FUNCTION fSHDLCChecksum : BYTE
VAR_INPUT
	i_bAdr	:	BYTE;
	i_bCmd	:	BYTE;
	i_bLen	:	BYTE;
	i_pbaTxData	:	POINTER TO BYTE;	
END_VAR
VAR
	iIndex	:	INT;
END_VAR

(* Checksum is calc like so
Sum all the bytes within the frame
Take the LSN ie. nibble of the result and invert it
*)

fSHDLCChecksum := i_bAdr + i_bCmd + i_bLen;

IF i_bLen > 0 THEN
FOR iIndex:=0 TO BYTE_TO_INT(i_bLen)DO
	fSHDLCChecksum := fSHDLCChecksum + i_pbaTxData^;
	i_pbaTxData := i_pbaTxData + 1;
END_FOR
END_IF

// Inverting LSN
fSHDLCChecksum := fSHDLCChecksum XOR 16#FF;

END_FUNCTION

(* stored: Version 1.1.0.1, ProductVersion 3.1.0.24
   POU fSHDLCChecksum: Id {a9b3b4d5-8205-40aa-be47-6f11775318a7} *)
